// TIA Portal V20 export
TYPE "Pallet"
   STRUCT
      IsSelected : Bool;
      "Name" : String;
      Station_Current_Position : Array[1..2] of Int;
      Number_Of_Elements : Array[1..4] of Int;
   END_STRUCT;
END_TYPE
